VAR_GLOBAL
END_VAR

(* stored: Version 1.1.0.1, ProductVersion 3.1.4024.12
   GVL GVL_ADS: Id {e84ef06f-0772-4e9d-ae4c-620ea62ec313} *)
